{attribute 'qualified_only'}
VAR_GLOBAL
END_VAR

(* stored: Version 1.1.0.1, ProductVersion 3.1.4024.4
   GVL Automatic: Id {a0828ab4-5402-4cb5-a4e0-5b8f242104b3} *)
